// TIA Portal V17 export
// export: Created 2022-03-14T21:17:28.4381403Z, ExportSetting WithDefaults, DisplayName Totally Integrated Automation Portal, DisplayVersion V17, DisplayName TIA Portal Openness, DisplayVersion V17, DisplayName TIA Portal Version Control Interface, DisplayVersion V17, DisplayName STEP 7 Professional, DisplayVersion V17, DisplayName STEP 7 Safety, DisplayVersion V17, DisplayName WinCC Advanced / Unified PC, DisplayVersion V17
FUNCTION_BLOCK "EM01_CM02_Palletizer"   // FB31672, LAD
TITLE = EM01_CM02
{ S7_Optimized_Access := 'TRUE' }
AUTHOR : tech.team.motioncontrol@siemens.com
FAMILY : CPG
VERSION : 1.1
// Support: tech.team.motioncontrol@siemens.com
// stored: AutoNumber true, IsIECCheckEnabled false, IsRetainMemResEnabled false, MemoryReserve 100, SetENOAutomatically false, UDAEnableTagReadback false
   VAR
      statDummyBool { ExternalAccessible := 'False'; ExternalVisible := 'False'; ExternalWritable := 'False'} : Bool;   // dummy bool - placeholder
      instPalletizer { S7_SetPoint := 'True'} : "Palletizer";
      Ntrig : Bool;
   END_VAR
   VAR_TEMP   // added for the SCL form of the ladder/FBD networks
      _w1 : Bool;
   END_VAR
BEGIN

REGION Network 1: *** Begin the Setpoint Management Information Section ***
END_REGION

REGION Network 2: *** Begin the Logic Section ***
END_REGION

REGION Network 3: Palletizer instance
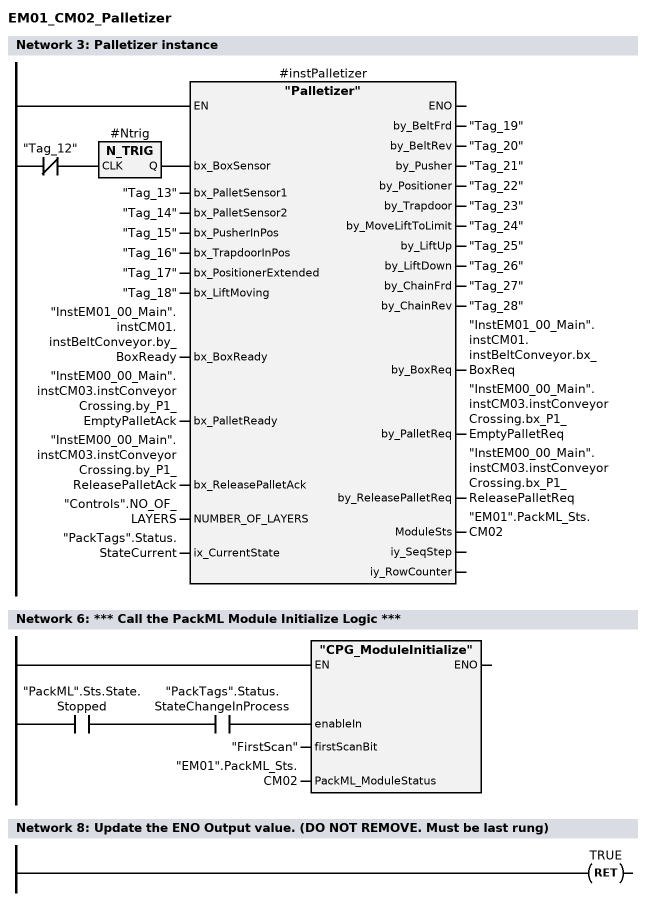
   RUNG wire#powerrail
      #instPalletizer(bx_BoxSensor := wire#w1, bx_PalletSensor1 := "Tag_13", bx_PalletSensor2 := "Tag_14", bx_PusherInPos := "Tag_15", bx_TrapdoorInPos := "Tag_16", bx_PositionerExtended := "Tag_17", bx_LiftMoving := "Tag_18", bx_BoxReady := "InstEM01_00_Main".instCM01.instBeltConveyor.by_BoxReady, bx_PalletReady := "InstEM00_00_Main".instCM03.instConveyorCrossing.by_P1_EmptyPalletAck, bx_ReleasePalletAck := "InstEM00_00_Main".instCM03.instConveyorCrossing.by_P1_ReleasePalletAck, NUMBER_OF_LAYERS := "Controls".NO_OF_LAYERS, ix_CurrentState := "PackTags".Status.StateCurrent, by_BeltFrd => "Tag_19", by_BeltRev => "Tag_20", by_Pusher => "Tag_21", by_Positioner => "Tag_22", by_Trapdoor => "Tag_23", by_MoveLiftToLimit => "Tag_24", by_LiftUp => "Tag_25", by_LiftDown => "Tag_26", by_ChainFrd => "Tag_27", by_ChainRev => "Tag_28", by_BoxReq => "InstEM01_00_Main".instCM01.instBeltConveyor.bx_BoxReq, by_PalletReq => "InstEM00_00_Main".instCM03.instConveyorCrossing.bx_P1_EmptyPalletReq, by_ReleasePalletReq => "InstEM00_00_Main".instCM03.instConveyorCrossing.bx_P1_ReleasePalletReq, ModuleSts => "EM01".PackML_Sts.CM02, iy_SeqStep =>, iy_RowCounter =>)
   END_RUNG
   RUNG wire#powerrail
      I_Contact( "Tag_12" )
      N_Trig( #Ntrig )
   END_RUNG wire#w1
   // the same network as SCL:
   #_w1 := NOT (NOT "Tag_12") AND #Ntrig;   // falling edge
   #Ntrig := NOT "Tag_12";
   #instPalletizer(bx_BoxSensor := #_w1,   // "Palletizer"
                   bx_PalletSensor1 := "Tag_13",
                   bx_PalletSensor2 := "Tag_14",
                   bx_PusherInPos := "Tag_15",
                   bx_TrapdoorInPos := "Tag_16",
                   bx_PositionerExtended := "Tag_17",
                   bx_LiftMoving := "Tag_18",
                   bx_BoxReady := "InstEM01_00_Main".instCM01.instBeltConveyor.by_BoxReady,
                   bx_PalletReady := "InstEM00_00_Main".instCM03.instConveyorCrossing.by_P1_EmptyPalletAck,
                   bx_ReleasePalletAck := "InstEM00_00_Main".instCM03.instConveyorCrossing.by_P1_ReleasePalletAck,
                   NUMBER_OF_LAYERS := "Controls".NO_OF_LAYERS,
                   ix_CurrentState := "PackTags".Status.StateCurrent,
                   by_BeltFrd => "Tag_19",
                   by_BeltRev => "Tag_20",
                   by_Pusher => "Tag_21",
                   by_Positioner => "Tag_22",
                   by_Trapdoor => "Tag_23",
                   by_MoveLiftToLimit => "Tag_24",
                   by_LiftUp => "Tag_25",
                   by_LiftDown => "Tag_26",
                   by_ChainFrd => "Tag_27",
                   by_ChainRev => "Tag_28",
                   by_BoxReq => "InstEM01_00_Main".instCM01.instBeltConveyor.bx_BoxReq,
                   by_PalletReq => "InstEM00_00_Main".instCM03.instConveyorCrossing.bx_P1_EmptyPalletReq,
                   by_ReleasePalletReq => "InstEM00_00_Main".instCM03.instConveyorCrossing.bx_P1_ReleasePalletReq,
                   ModuleSts => "EM01".PackML_Sts.CM02);
END_REGION

REGION Network 4: *** Begin the Event Information Section ***
END_REGION

REGION Network 5: *** Begin the State Model Status Feedback Section ***
END_REGION

REGION Network 6: *** Call the PackML Module Initialize Logic ***
   RUNG wire#powerrail
      "CPG_ModuleInitialize"(enableIn := wire#w1, firstScanBit := "FirstScan", PackML_ModuleStatus := "EM01".PackML_Sts.CM02)
   END_RUNG
   RUNG wire#powerrail
      Contact( "PackML".Sts.State.Stopped )
      Contact( "PackTags".Status.StateChangeInProcess )
   END_RUNG wire#w1
   // the same network as SCL:
   "CPG_ModuleInitialize"(enableIn := "PackML".Sts.State.Stopped AND "PackTags".Status.StateChangeInProcess,
                          firstScanBit := "FirstScan",
                          PackML_ModuleStatus := "EM01".PackML_Sts.CM02);
END_REGION

REGION Network 8: Update the ENO Output value. (DO NOT REMOVE. Must be last rung)
   RUNG wire#powerrail
      ReturnCoil( TRUE )
   END_RUNG
   // the same network as SCL:
   ENO := TRUE;
   RETURN;
END_REGION
END_FUNCTION_BLOCK
